{attribute 'GeneratedUsingTerminal: EL3314-0030-0021'}
{attribute addProperty BoxType "EL3314-0030-0021"}
{attribute addProperty Id "StatusAT %I*Status_68C33E995ValueAT %I*DINT4"}
{attribute addProperty CRC "542107472"}
{attribute addProperty Size "9"}
TYPE TC_Inputs_Channel_204FE750 EXTENDS InputBase_8311D824 :
STRUCT
	{attribute addProperty Name "Status"}
	Status AT %I* : Status_68C33E99;
	{attribute addProperty Name "Value"}
	Value AT %I* : DINT;
END_STRUCT
END_TYPE

(* stored: Version 1.2.0.0, ProductVersion 3.1.4024.11
   DUT TC_Inputs_Channel_204FE750: Id {c41e638f-3282-48ab-beed-ae23fe9826b0} *)
